(* Logix 5000 project; controller PLC_ABB vendor 1 type 14 code 77 rev 20.11; software revision 20.00 *)

TASK MainTask (continuous, watchdog 500 ms) : MainProgram

MODULES
   Controller : vendor 1 type 14 code 77 (CompactLogixL32EController 0, rev 20.11)
      LocalENB : 1769-L32E Ethernet Port (CompactLogixL32Ethernet 1, rev 20.11)
         PLC_DC : 1769-L32E Ethernet Port (Ethernet 192.168.2.131, rev 20.1)
            PLC_DC_Controller : vendor 1 type 14 code 77 (CompactLogixL32EController 0, rev 20.1, $a7c5510e$ RPI 20 ms, $928fdd19$ RPI 20 ms, $93e49bd8$ RPI 20 ms)
         ABBDrive : ETHERNET-MODULE (Ethernet 192.168.2.40, rev 1.1, Output RPI 20 ms)
      Local : CompactBus (CompactVirtualAdapter 3, rev 20.11)
         IO_Digital_Module : vendor 1 type 7 code 66 (Compact 2, rev 2.1, Output RPI 20 ms)
         hartModule : vendor 58 type 10 code 4 (Compact 1, rev 3.1, Output RPI 80 ms)
END_MODULES

TYPE ABB_Read :
STRUCT
   Logic_Status_Word : LSW;
   RPM_Feedback : INT;
   RPM_Referencia : INT;
   Output_Power : REAL;
   BusDC : REAL;
   Output_Current : REAL;
   Output_Voltage : REAL;
   PF : REAL;
   Latest_Fault : INT;
   Accel : BOOL;
   Descell : BOOL;
   PercentTemperature : INT;
END_STRUCT
END_TYPE

TYPE ABB_Write :
STRUCT
   RPM_Reference : INT;
   Run_Forward : BOOL;
   Run_Reverse : BOOL;
   Reset_Fault : BOOL;
END_STRUCT
END_TYPE

TYPE ComandVSD :
STRUCT
   start : BOOL;
   stop : BOOL;
   reset : BOOL;
   referencia : REAL;
   direction : BOOL;
END_STRUCT
END_TYPE

TYPE Dinagrama :
STRUCT
   vPotencia : REAL[500];
   vCarga : REAL[500];
   vPosicion : REAL[500];
   vProximetro : DINT[500];
   NumeroMuestras : INT;
   enabled : BOOL;
   captura : BOOL;
   resetVector : BOOL;
   vEmptyREAL : REAL[500];
   vEmptyINT : DINT[500];
   tMuestreo : REAL;
END_STRUCT
END_TYPE

TYPE ethImplicitRead :
STRUCT
   Enabled : BOOL;
   Done : BOOL;
   Error : BOOL;
   Value : DINT;
   instance : DINT;
   atribute : INT;
END_STRUCT
END_TYPE

TYPE ethImplicitWrite :
STRUCT
   Enabled : BOOL;
   Done : BOOL;
   ERR : BOOL;
   Value : DINT;
   Instance : DINT;
   Atribute : INT;
   clase : INT;
END_STRUCT
END_TYPE

TYPE LSW :
STRUCT
   Faulted : BOOL;
   Warning : BOOL;
   RunForward : BOOL;
   RunReverse : BOOL;
   Ready : BOOL;
   RemoteRef : BOOL;
   RemoteCrtl : BOOL;
   AtSpeed : BOOL;
END_STRUCT
END_TYPE

TYPE SWC :
STRUCT
   comand : ComandVSD;
   Dinagrama : Dinagrama;
   entradasDigitales : INT;
   salidasDigitales : INT;
   entradasAnalogas : REAL[4];
   salidasAnalogas : REAL[4];
   ABBRead : ABB_Read;
   etheWrite : ethImplicitWrite;
   etheRead : ethImplicitRead;
END_STRUCT
END_TYPE

TYPE VSD :
STRUCT
   LogicCommand_Start : BOOL;
   LogicCommand_Stop : BOOL;
   LogicCommand_ClearFaults : BOOL;
   LogicCommand_Forward : BOOL;
   LogicCommand_Reverse : BOOL;
   Reference : REAL;
END_STRUCT
END_TYPE

VAR_GLOBAL   (* controller tags *)
   ABB_GetAtt_Value : DINT := 7500;
   ABB_GetMsg : MESSAGE;
        MessageParameters(ServiceCode := 16#000e, DestinationTag := ABB_GetAtt_Value, ...)
   ABB_Input : ABB_Read := (Logic_Status_Word.Ready := 1, Logic_Status_Word.RemoteRef := 1, Logic_Status_Word.RemoteCrtl := 1, RPM_Referencia := 180, Output_Power := 5.8945793e-37, BusDC := 678.1, Latest_Fault := 8976, PercentTemperature := 20);
   ABB_Msg_SetValue : DINT := 60000;
   ABB_Output : ABB_Write := (RPM_Reference := 180);
   ABB_SetMsg : MESSAGE;
        MessageParameters(ServiceCode := 16#0010, LocalElement := ABB_Msg_SetValue, ...)
   Proximetro : BOOL;
   SRP_Displacement_Actual : REAL := 0.643343;
   SRP_Load_Actual : REAL := 9.741267;
   SRP_SimActualStroke : DINT := 1;
   SWC : SWC := (comand.referencia := 180.0, comand.direction := 1, Dinagrama.vPotencia[0] := 5.890374e-37, Dinagrama.vPotencia[1] := 5.890374e-37, Dinagrama.vPotencia[2] := 5.890374e-37, Dinagrama.vPotencia[3] := 5.890374e-37, Dinagrama.vPotencia[4] := 5.890374e-37, Dinagrama.vPotencia[5] := 5.890374e-37, Dinagrama.vPotencia[6] := 5.890374e-37, Dinagrama.vPotencia[7] := 5.890374e-37, Dinagrama.vPotencia[8] := 5.890374e-37, Dinagrama.vPotencia[9] := 5.890374e-37, Dinagrama.vPotencia[10] := 5.890374e-37, Dinagrama.vPotencia[11] := 5.890374e-37, Dinagrama.vPotencia[12] := 5.890374e-37, Dinagrama.vPotencia[13] := 5.890374e-37, Dinagrama.vPotencia[14] := 5.890374e-37, Dinagrama.vPotencia[15] := 5.890374e-37, Dinagrama.vPotencia[16] := 5.890374e-37, Dinagrama.vPotencia[17] := 5.890374e-37, Dinagrama.vPotencia[18] := 5.890374e-37, Dinagrama.vPotencia[19] := 5.890374e-37, Dinagrama.vPotencia[20] := 5.890374e-37, Dinagrama.vPotencia[21] := 5.890374e-37, Dinagrama.vPotencia[22] := 5.890374e-37, Dinagrama.vPotencia[23] := 5.890374e-37, Dinagrama.vPotencia[24] := 5.890374e-37, Dinagrama.vPotencia[25] := 5.890374e-37, Dinagrama.vPotencia[26] := 5.890374e-37, Dinagrama.vPotencia[27] := 5.890374e-37, Dinagrama.vPotencia[28] := 5.890374e-37, Dinagrama.vPotencia[29] := 5.890374e-37, Dinagrama.vPotencia[30] := 5.890374e-37, Dinagrama.vPotencia[31] := 5.890374e-37, Dinagrama.vPotencia[32] := 5.890374e-37, Dinagrama.vPotencia[33] := 5.890374e-37, Dinagrama.vPotencia[34] := 5.890374e-37, Dinagrama.vPotencia[35] := 5.890374e-37, Dinagrama.vPotencia[36] := 5.890374e-37, Dinagrama.vPotencia[37] := 5.890374e-37, Dinagrama.vPotencia[38] := 5.890374e-37, Dinagrama.vPotencia[39] := 5.890374e-37, Dinagrama.vPotencia[40] := 5.890374e-37, Dinagrama.vPotencia[41] := 5.890374e-37, Dinagrama.vPotencia[42] := 5.890374e-37, Dinagrama.vPotencia[43] := 5.890374e-37, Dinagrama.vPotencia[44] := 5.890374e-37, Dinagrama.vPotencia[45] := 5.890374e-37, Dinagrama.vPotencia[46] := 5.890374e-37, Dinagrama.vPotencia[47] := 5.890374e-37, Dinagrama.vPotencia[48] := 5.890374e-37, Dinagrama.vPotencia[49] := 5.890374e-37, Dinagrama.vPotencia[50] := 5.890374e-37, Dinagrama.vPotencia[51] := 5.890374e-37, Dinagrama.vPotencia[52] := 5.890374e-37, Dinagrama.vPotencia[53] := 5.890374e-37, Dinagrama.vPotencia[54] := 5.890374e-37, Dinagrama.vPotencia[55] := 5.890374e-37, Dinagrama.vPotencia[56] := 5.890374e-37, Dinagrama.vPotencia[57] := 5.890374e-37,
        Dinagrama.vPotencia[58] := 5.890374e-37, Dinagrama.vPotencia[59] := 5.890374e-37, Dinagrama.vPotencia[60] := 5.890374e-37, Dinagrama.vPotencia[61] := 5.890374e-37, Dinagrama.vPotencia[62] := 5.890374e-37, Dinagrama.vPotencia[63] := 5.890374e-37, Dinagrama.vPotencia[64] := 5.890374e-37, Dinagrama.vPotencia[65] := 5.890374e-37, Dinagrama.vPotencia[66] := 5.890374e-37, Dinagrama.vPotencia[67] := 5.890374e-37, Dinagrama.vPotencia[68] := 5.890374e-37, Dinagrama.vPotencia[69] := 5.890374e-37, Dinagrama.vPotencia[70] := 5.890374e-37, Dinagrama.vPotencia[71] := 5.890374e-37, Dinagrama.vPotencia[72] := 5.890374e-37, Dinagrama.vPotencia[73] := 5.890374e-37, Dinagrama.vPotencia[74] := 5.890374e-37, Dinagrama.vPotencia[75] := 5.890374e-37, Dinagrama.vPotencia[76] := 5.890374e-37, Dinagrama.vPotencia[77] := 5.890374e-37, Dinagrama.vPotencia[78] := 5.890374e-37, Dinagrama.vPotencia[79] := 5.890374e-37, Dinagrama.vPotencia[80] := 5.890374e-37, Dinagrama.vPotencia[81] := 5.890374e-37, Dinagrama.vPotencia[82] := 5.890374e-37, Dinagrama.vPotencia[83] := 5.890374e-37, Dinagrama.vPotencia[84] := 5.890374e-37, Dinagrama.vPotencia[85] := 5.890374e-37, Dinagrama.vPotencia[86] := 5.890374e-37, Dinagrama.vPotencia[87] := 5.890374e-37, Dinagrama.vPotencia[88] := 5.890374e-37, Dinagrama.vPotencia[89] := 5.890374e-37, Dinagrama.vPotencia[90] := 5.890374e-37, Dinagrama.vPotencia[91] := 5.890374e-37, Dinagrama.vPotencia[92] := 5.890374e-37, Dinagrama.vPotencia[93] := 5.890374e-37, Dinagrama.vPotencia[94] := 5.890374e-37, Dinagrama.vPotencia[95] := 5.890374e-37, Dinagrama.vPotencia[96] := 5.890374e-37, Dinagrama.vPotencia[97] := 5.890374e-37, Dinagrama.vPotencia[98] := 5.890374e-37, Dinagrama.vPotencia[99] := 5.890374e-37, Dinagrama.vPotencia[100] := 5.890374e-37, Dinagrama.vPotencia[101] := 5.890374e-37, Dinagrama.vPotencia[102] := 5.890374e-37, Dinagrama.vPotencia[103] := 5.890374e-37, Dinagrama.vPotencia[104] := 5.890374e-37, Dinagrama.vPotencia[105] := 5.890374e-37, Dinagrama.vPotencia[106] := 5.890374e-37, Dinagrama.vPotencia[107] := 5.890374e-37, Dinagrama.vPotencia[108] := 5.890374e-37, Dinagrama.vPotencia[109] := 5.890374e-37, Dinagrama.vPotencia[110] := 5.890374e-37, Dinagrama.vPotencia[111] := 5.890374e-37, Dinagrama.vPotencia[112] := 5.890374e-37, Dinagrama.vPotencia[113] := 5.890374e-37, Dinagrama.vPotencia[114] := 5.890374e-37, Dinagrama.vPotencia[115] := 5.890374e-37, Dinagrama.vPotencia[116] := 5.890374e-37, Dinagrama.vPotencia[117] := 5.890374e-37,
        Dinagrama.vPotencia[118] := 5.890374e-37, Dinagrama.vPotencia[119] := 5.890374e-37, Dinagrama.vPotencia[120] := 5.890374e-37, Dinagrama.vPotencia[121] := 5.890374e-37, Dinagrama.vPotencia[122] := 5.890374e-37, Dinagrama.vPotencia[123] := 5.890374e-37, Dinagrama.vPotencia[124] := 5.890374e-37, Dinagrama.vPotencia[125] := 5.890374e-37, Dinagrama.vPotencia[126] := 5.890374e-37, Dinagrama.vPotencia[127] := 5.890374e-37, Dinagrama.vPotencia[128] := 5.890374e-37, Dinagrama.vPotencia[129] := 5.890374e-37, Dinagrama.vPotencia[130] := 5.890374e-37, Dinagrama.vPotencia[131] := 5.890374e-37, Dinagrama.vPotencia[132] := 5.890374e-37, Dinagrama.vPotencia[133] := 5.890374e-37, Dinagrama.vPotencia[134] := 5.890374e-37, Dinagrama.vPotencia[135] := 5.890374e-37, Dinagrama.vPotencia[136] := 5.890374e-37, Dinagrama.vPotencia[137] := 5.890374e-37, Dinagrama.vPotencia[138] := 5.890374e-37, Dinagrama.vPotencia[139] := 5.890374e-37, Dinagrama.vPotencia[140] := 5.890374e-37, Dinagrama.vPotencia[141] := 5.890374e-37, Dinagrama.vPotencia[142] := 5.8988127e-37, Dinagrama.vCarga[0] := 9.6614, Dinagrama.vCarga[1] := 9.7812, Dinagrama.vCarga[2] := 9.711983, Dinagrama.vCarga[3] := 9.725293, Dinagrama.vCarga[4] := 9.842433, Dinagrama.vCarga[5] := 9.70932, Dinagrama.vCarga[6] := 9.69601, Dinagrama.vCarga[7] := 9.7306185, Dinagrama.vCarga[8] := 9.586858, Dinagrama.vCarga[9] := 9.751916, Dinagrama.vCarga[10] := 10.223133, Dinagrama.vCarga[11] := 10.473384, Dinagrama.vCarga[12] := 10.633119, Dinagrama.vCarga[13] := 10.856748, Dinagrama.vCarga[14] := 11.029794, Dinagrama.vCarga[15] := 11.220809, Dinagrama.vCarga[16] := 11.419147, Dinagrama.vCarga[17] := 11.515653, Dinagrama.vCarga[18] := 11.655421, Dinagrama.vCarga[19] := 11.805838, Dinagrama.vCarga[20] := 11.900348, Dinagrama.vCarga[21] := 11.940947, Dinagrama.vCarga[22] := 11.73795, Dinagrama.vCarga[23] := 11.4471, Dinagrama.vCarga[24] := 11.15625, Dinagrama.vCarga[25] := 10.976548, Dinagrama.vCarga[26] := 10.774218, Dinagrama.vCarga[27] := 10.571887, Dinagrama.vCarga[28] := 10.393517, Dinagrama.vCarga[29] := 10.257743, Dinagrama.vCarga[30] := 10.105995, Dinagrama.vCarga[31] := 10.018141, Dinagrama.vCarga[32] := 9.762565, Dinagrama.vCarga[33] := 9.634777, Dinagrama.vCarga[34] := 9.706658,
        Dinagrama.vCarga[35] := 9.826459, Dinagrama.vCarga[36] := 10.050088, Dinagrama.vCarga[37] := 10.177875, Dinagrama.vCarga[38] := 10.321636, Dinagrama.vCarga[39] := 10.409491, Dinagrama.vCarga[40] := 10.417477, Dinagrama.vCarga[41] := 10.401504, Dinagrama.vCarga[42] := 10.518642, Dinagrama.vCarga[43] := 10.481371, Dinagrama.vCarga[44] := 10.476047, Dinagrama.vCarga[45] := 10.63312, Dinagrama.vCarga[46] := 10.715649, Dinagrama.vCarga[47] := 10.476047, Dinagrama.vCarga[48] := 10.17255, Dinagrama.vCarga[49] := 9.970221, Dinagrama.vCarga[50] := 9.850419, Dinagrama.vCarga[51] := 9.608155, Dinagrama.vCarga[52] := 9.397838, Dinagrama.vCarga[53] := 9.405825, Dinagrama.vCarga[54] := 9.34193, Dinagrama.vCarga[55] := 9.131613, Dinagrama.vCarga[56] := 9.049084, Dinagrama.vCarga[57] := 9.08103, Dinagrama.vCarga[58] := 8.9266205, Dinagrama.vCarga[59] := 8.873376, Dinagrama.vCarga[60] := 9.155573, Dinagrama.vCarga[61] := 9.427122, Dinagrama.vCarga[62] := 9.549585, Dinagrama.vCarga[63] := 9.682697, Dinagrama.vCarga[64] := 9.906326, Dinagrama.vCarga[65] := 10.012816, Dinagrama.vCarga[66] := 9.980869, Dinagrama.vCarga[67] := 9.986194, Dinagrama.vCarga[68] := 9.962234, Dinagrama.vCarga[69] := 10.018141, Dinagrama.vCarga[70] := 10.042101, Dinagrama.vCarga[71] := 10.098008, Dinagrama.vCarga[72] := 10.193849, Dinagrama.vCarga[73] := 9.938273, Dinagrama.vCarga[74] := 9.618804, Dinagrama.vCarga[75] := 9.546924, Dinagrama.vCarga[76] := 9.55491, Dinagrama.vCarga[77] := 9.331282, Dinagrama.vCarga[78] := 9.171547, Dinagrama.vCarga[79] := 9.347255, Dinagrama.vCarga[80] := 9.219467, Dinagrama.vCarga[81] := 9.123626, Dinagrama.vCarga[82] := 9.18752, Dinagrama.vCarga[83] := 9.331282, Dinagrama.vCarga[84] := 9.166222, Dinagrama.vCarga[85] := 9.400499, Dinagrama.vCarga[86] := 9.565559, Dinagrama.vCarga[87] := 9.762566, Dinagrama.vCarga[88] := 9.688023, Dinagrama.vCarga[89] := 9.746592, Dinagrama.vCarga[90] := 9.885028, Dinagrama.vCarga[91] := 9.834445, Dinagrama.vCarga[92] := 9.634777, Dinagrama.vCarga[93] := 9.640101, Dinagrama.vCarga[94] := 9.624128,
        Dinagrama.vCarga[95] := 9.37654, Dinagrama.vCarga[96] := 9.184858, Dinagrama.vCarga[97] := 9.046422, Dinagrama.vCarga[98] := 8.665721, Dinagrama.vCarga[99] := 8.223788, Dinagrama.vCarga[100] := 7.936266, Dinagrama.vCarga[101] := 7.851074, Dinagrama.vCarga[102] := 7.6647167, Dinagrama.vCarga[103] := 7.398492, Dinagrama.vCarga[104] := 7.281353, Dinagrama.vCarga[105] := 7.238757, Dinagrama.vCarga[106] := 6.993831, Dinagrama.vCarga[107] := 6.706309, Dinagrama.vCarga[108] := 6.6796865, Dinagrama.vCarga[109] := 6.903315, Dinagrama.vCarga[110] := 7.1056457, Dinagrama.vCarga[111] := 7.3771944, Dinagrama.vCarga[112] := 7.773869, Dinagrama.vCarga[113] := 7.91763, Dinagrama.vCarga[114] := 7.909643, Dinagrama.vCarga[115] := 7.909643, Dinagrama.vCarga[116] := 8.300993, Dinagrama.vCarga[117] := 8.340926, Dinagrama.vCarga[118] := 8.460728, Dinagrama.vCarga[119] := 8.596502, Dinagrama.vCarga[120] := 8.804157, Dinagrama.vCarga[121] := 8.788184, Dinagrama.vCarga[122] := 8.77221, Dinagrama.vCarga[123] := 8.588515, Dinagrama.vCarga[124] := 8.420794, Dinagrama.vCarga[125] := 8.340927, Dinagrama.vCarga[126] := 8.468715, Dinagrama.vCarga[127] := 8.431443, Dinagrama.vCarga[128] := 8.476701, Dinagrama.vCarga[129] := 8.580528, Dinagrama.vCarga[130] := 8.497999, Dinagrama.vCarga[131] := 8.503324, Dinagrama.vCarga[132] := 8.575204, Dinagrama.vCarga[133] := 8.56988, Dinagrama.vCarga[134] := 8.631111, Dinagrama.vCarga[135] := 8.84409, Dinagrama.vCarga[136] := 9.081031, Dinagrama.vCarga[137] := 9.278037, Dinagrama.vCarga[138] := 9.325957, Dinagrama.vCarga[139] := 9.363229, Dinagrama.vCarga[140] := 9.618804, Dinagrama.vCarga[141] := 9.682698, Dinagrama.vCarga[142] := 9.682698, Dinagrama.vPosicion[0] := 0.0550175, Dinagrama.vPosicion[1] := 0.4084145, Dinagrama.vPosicion[2] := 0.8989175, Dinagrama.vPosicion[3] := 1.5143573, Dinagrama.vPosicion[4] := 2.2604218, Dinagrama.vPosicion[5] := 3.6340683, Dinagrama.vPosicion[6] := 4.147569, Dinagrama.vPosicion[7] := 5.2654533, Dinagrama.vPosicion[8] := 6.4805126, Dinagrama.vPosicion[9] := 7.78114, Dinagrama.vPosicion[10] := 9.158964, Dinagrama.vPosicion[11] := 10.613574,
        Dinagrama.vPosicion[12] := 12.155543, Dinagrama.vPosicion[13] := 13.778378, Dinagrama.vPosicion[14] := 15.740422, Dinagrama.vPosicion[15] := 17.481466, Dinagrama.vPosicion[16] := 19.2797, Dinagrama.vPosicion[17] := 21.118301, Dinagrama.vPosicion[18] := 22.99865, Dinagrama.vPosicion[19] := 24.928076, Dinagrama.vPosicion[20] := 26.89821, Dinagrama.vPosicion[21] := 28.908155, Dinagrama.vPosicion[22] := 30.958275, Dinagrama.vPosicion[23] := 33.057575, Dinagrama.vPosicion[24] := 35.193996, Dinagrama.vPosicion[25] := 37.35984, Dinagrama.vPosicion[26] := 39.561394, Dinagrama.vPosicion[27] := 41.798325, Dinagrama.vPosicion[28] := 44.44635, Dinagrama.vPosicion[29] := 46.757927, Dinagrama.vPosicion[30] := 49.113125, Dinagrama.vPosicion[31] := 50.300934, Dinagrama.vPosicion[32] := 53.71554, Dinagrama.vPosicion[33] := 56.007725, Dinagrama.vPosicion[34] := 58.29858, Dinagrama.vPosicion[35] := 59.435463, Dinagrama.vPosicion[36] := 61.651955, Dinagrama.vPosicion[37] := 64.96143, Dinagrama.vPosicion[38] := 67.1463, Dinagrama.vPosicion[39] := 69.277466, Dinagrama.vPosicion[40] := 70.327156, Dinagrama.vPosicion[41] := 72.39657, Dinagrama.vPosicion[42] := 74.763824, Dinagrama.vPosicion[43] := 77.68309, Dinagrama.vPosicion[44] := 78.62532, Dinagrama.vPosicion[45] := 80.46515, Dinagrama.vPosicion[46] := 82.25429, Dinagrama.vPosicion[47] := 83.99117, Dinagrama.vPosicion[48] := 85.65761, Dinagrama.vPosicion[49] := 87.23202, Dinagrama.vPosicion[50] := 88.73018, Dinagrama.vPosicion[51] := 90.154045, Dinagrama.vPosicion[52] := 91.48115, Dinagrama.vPosicion[53] := 92.103096, Dinagrama.vPosicion[54] := 93.858185, Dinagrama.vPosicion[55] := 94.9114, Dinagrama.vPosicion[56] := 96.00089, Dinagrama.vPosicion[57] := 96.84068, Dinagrama.vPosicion[58] := 97.581314, Dinagrama.vPosicion[59] := 98.21293, Dinagrama.vPosicion[60] := 98.7474, Dinagrama.vPosicion[61] := 99.18755, Dinagrama.vPosicion[62] := 99.53332, Dinagrama.vPosicion[63] := 99.672134, Dinagrama.vPosicion[64] := 99.935196, Dinagrama.vPosicion[65] := 99.99795, Dinagrama.vPosicion[66] := 99.96849, Dinagrama.vPosicion[67] := 99.8579, Dinagrama.vPosicion[68] := 99.76811, Dinagrama.vPosicion[69] := 99.35959, Dinagrama.vPosicion[70] := 98.93282, Dinagrama.vPosicion[71] := 98.72924,
        Dinagrama.vPosicion[72] := 98.26827, Dinagrama.vPosicion[73] := 97.74029, Dinagrama.vPosicion[74] := 97.14606, Dinagrama.vPosicion[75] := 96.147736, Dinagrama.vPosicion[76] := 95.795845, Dinagrama.vPosicion[77] := 95.004196, Dinagrama.vPosicion[78] := 94.16693, Dinagrama.vPosicion[79] := 93.305756, Dinagrama.vPosicion[80] := 91.870316, Dinagrama.vPosicion[81] := 91.377556, Dinagrama.vPosicion[82] := 90.37801, Dinagrama.vPosicion[83] := 89.32036, Dinagrama.vPosicion[84] := 87.43099, Dinagrama.vPosicion[85] := 86.2471, Dinagrama.vPosicion[86] := 85.63856, Dinagrama.vPosicion[87] := 84.37339, Dinagrama.vPosicion[88] := 83.06744, Dinagrama.vPosicion[89] := 81.722916, Dinagrama.vPosicion[90] := 79.59406, Dinagrama.vPosicion[91] := 78.86634, Dinagrama.vPosicion[92] := 77.38295, Dinagrama.vPosicion[93] := 75.84359, Dinagrama.vPosicion[94] := 74.24831, Dinagrama.vPosicion[95] := 72.63172, Dinagrama.vPosicion[96] := 70.97654, Dinagrama.vPosicion[97] := 69.25514, Dinagrama.vPosicion[98] := 67.223434, Dinagrama.vPosicion[99] := 65.45152, Dinagrama.vPosicion[100] := 63.614063, Dinagrama.vPosicion[101] := 61.744232, Dinagrama.vPosicion[102] := 59.862404, Dinagrama.vPosicion[103] := 57.93054, Dinagrama.vPosicion[104] := 55.949615, Dinagrama.vPosicion[105] := 53.960396, Dinagrama.vPosicion[106] := 51.950417, Dinagrama.vPosicion[107] := 49.88953, Dinagrama.vPosicion[108] := 47.795254, Dinagrama.vPosicion[109] := 45.690845, Dinagrama.vPosicion[110] := 43.56501, Dinagrama.vPosicion[111] := 41.413986, Dinagrama.vPosicion[112] := 38.891975, Dinagrama.vPosicion[113] := 36.722637, Dinagrama.vPosicion[114] := 34.528854, Dinagrama.vPosicion[115] := 33.423225, Dinagrama.vPosicion[116] := 30.155361, Dinagrama.vPosicion[117] := 27.987307, Dinagrama.vPosicion[118] := 25.821117, Dinagrama.vPosicion[119] := 24.743301, Dinagrama.vPosicion[120] := 22.634195, Dinagrama.vPosicion[121] := 20.581553, Dinagrama.vPosicion[122] := 17.632542, Dinagrama.vPosicion[123] := 15.761359, Dinagrama.vPosicion[124] := 14.84577, Dinagrama.vPosicion[125] := 13.085015, Dinagrama.vPosicion[126] := 11.154951, Dinagrama.vPosicion[127] := 8.857708, Dinagrama.vPosicion[128] := 8.136012, Dinagrama.vPosicion[129] := 6.7788615, Dinagrama.vPosicion[130] := 5.529149, Dinagrama.vPosicion[131] := 4.3940463,
        Dinagrama.vPosicion[132] := 2.945591, Dinagrama.vPosicion[133] := 2.520764, Dinagrama.vPosicion[134] := 1.7710685, Dinagrama.vPosicion[135] := 1.148738, Dinagrama.vPosicion[136] := 0.66532767, Dinagrama.vPosicion[137] := 0.31461334, Dinagrama.vPosicion[138] := 0.096083336, Dinagrama.vPosicion[139] := 0.009929333, Dinagrama.vPosicion[140] := 0.049646668, Dinagrama.vPosicion[141] := 0.059576, Dinagrama.vPosicion[142] := 0.059576, Dinagrama.vProximetro[0] := 1, Dinagrama.vProximetro[1] := 1, Dinagrama.vProximetro[2] := 1, Dinagrama.NumeroMuestras := 141, Dinagrama.tMuestreo := 0.05, entradasAnalogas[0] := 16.901644, entradasAnalogas[1] := 13.587194, entradasAnalogas[2] := 3.2056525, entradasAnalogas[3] := 3.2056525, ABBRead.Logic_Status_Word.Ready := 1, ABBRead.Logic_Status_Word.RemoteRef := 1, ABBRead.Logic_Status_Word.RemoteCrtl := 1, ABBRead.RPM_Referencia := 180, ABBRead.Output_Power := 5.8945793e-37, ABBRead.BusDC := 678.1, ABBRead.Latest_Fault := 8976, ABBRead.PercentTemperature := 20, etheWrite.Enabled := 1, etheWrite.ERR := 1, etheWrite.Value := 60000, etheWrite.Instance := 23, etheWrite.Atribute := 13, etheRead.Value := 7500, etheRead.instance := 99, etheRead.atribute := 10);
   Timmers : TIMER[10] := ([0].PRE := 43, [1].PRE := 828000, [1].ACC := 352537, [1].EN := 1, [1].TT := 1, [2].PRE := 500, [3].PRE := 1000, [4].PRE := 10000);
END_VAR

PROGRAM MainProgram   (* main routine R000_MainRoutine *)
VAR
   Captura : BOOL;
   contadorAux : ALIAS FOR counter[0].ACC;
   counter : COUNTER[10];
   Flag : BOOL;
   flagDesAcell : BOOL;
   myoneshot : BOOL[32] := ([0] := 1);
   Proximetro_Virtual : ALIAS FOR SRP_SimActualStroke;
   rpmFeedback : INT;
   SPM_Reference : REAL := 8.5;
   timer : TIMER[10] := ([0].PRE := 50);
END_VAR

ROUTINE R000_MainRoutine   (* ladder *)
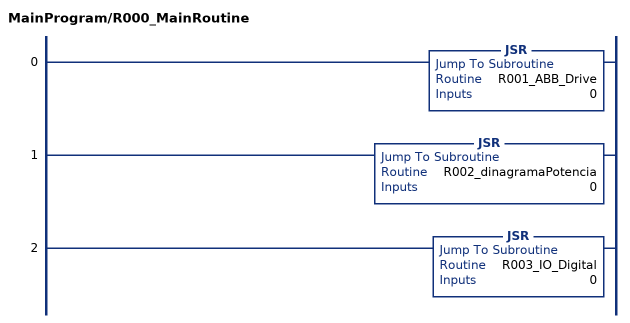
   0: JSR(R001_ABB_Drive,0);
   1: JSR(R002_dinagramaPotencia,0);
   2: JSR(R003_IO_Digital,0);
END_ROUTINE

ROUTINE R001_ABB_Drive   (* ladder *)
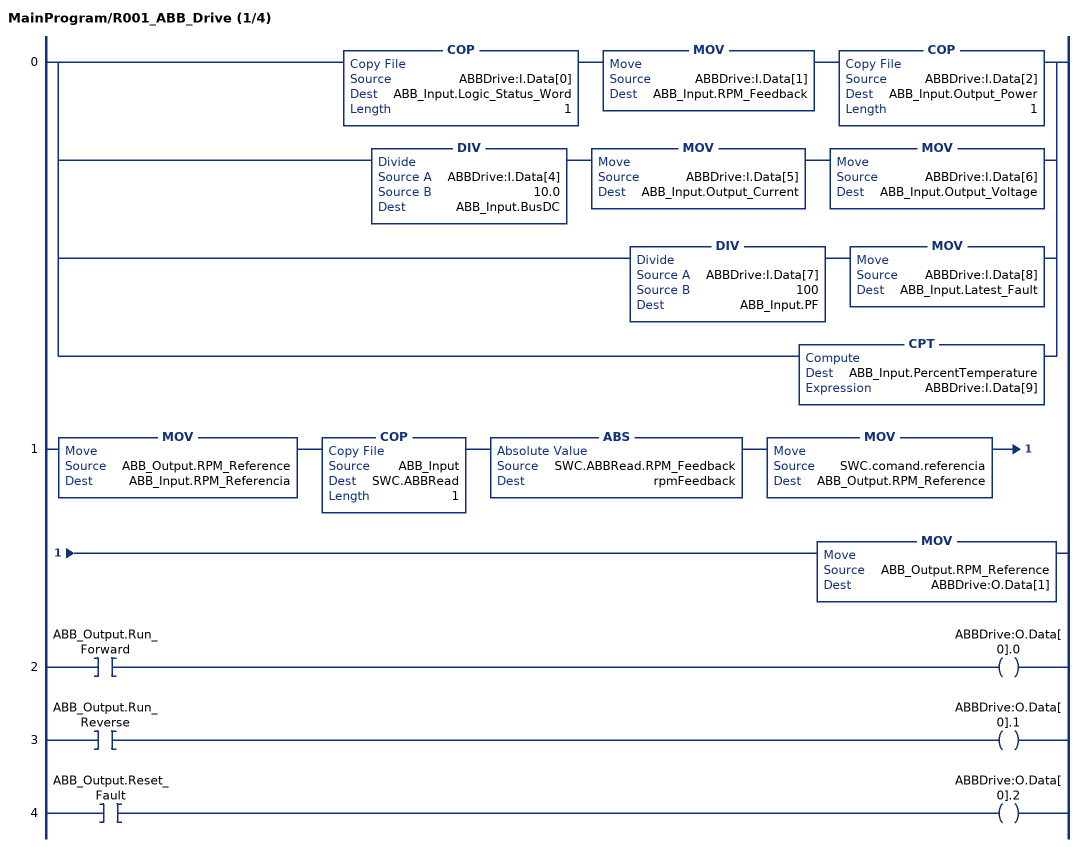
   0: [COP(ABBDrive:I.Data[0],ABB_Input.Logic_Status_Word,1) MOV(ABBDrive:I.Data[1],ABB_Input.RPM_Feedback) COP(ABBDrive:I.Data[2],ABB_Input.Output_Power,1) ,DIV(ABBDrive:I.Data[4],10.0,ABB_Input.BusDC) MOV(ABBDrive:I.Data[5],ABB_Input.Output_Current) MOV(ABBDrive:I.Data[6],ABB_Input.Output_Voltage) ,[DIV(ABBDrive:I.Data[7],100,ABB_Input.PF) MOV(ABBDrive:I.Data[8],ABB_Input.Latest_Fault) ,CPT(ABB_Input.PercentTemperature,ABBDrive:I.Data[9]) ] ];
   1: MOV(ABB_Output.RPM_Reference,ABB_Input.RPM_Referencia)COP(ABB_Input,SWC.ABBRead,1)ABS(SWC.ABBRead.RPM_Feedback,rpmFeedback)MOV(SWC.comand.referencia,ABB_Output.RPM_Reference)MOV(ABB_Output.RPM_Reference,ABBDrive:O.Data[1]);
   2: XIC(ABB_Output.Run_Forward)OTE(ABBDrive:O.Data[0].0);
   3: XIC(ABB_Output.Run_Reverse)OTE(ABBDrive:O.Data[0].1);
   4: XIC(ABB_Output.Reset_Fault)OTE(ABBDrive:O.Data[0].2);
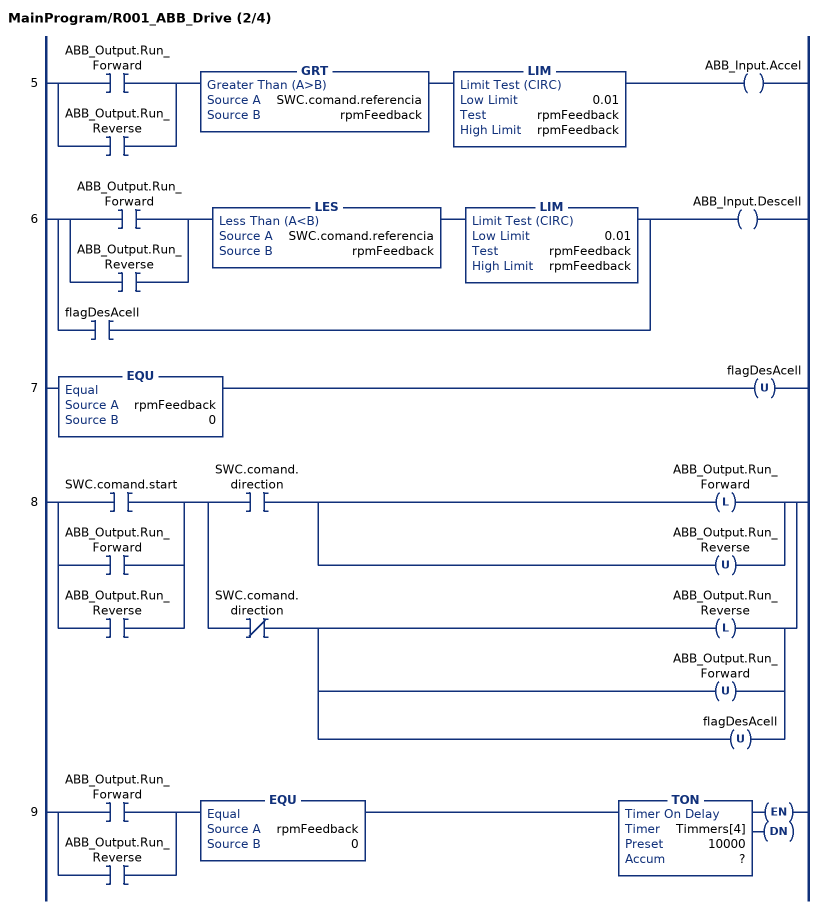
   5: [XIC(ABB_Output.Run_Forward) ,XIC(ABB_Output.Run_Reverse) ]GRT(SWC.comand.referencia,rpmFeedback)LIM(0.01,rpmFeedback,rpmFeedback)OTE(ABB_Input.Accel);
   6: [[XIC(ABB_Output.Run_Forward) ,XIC(ABB_Output.Run_Reverse) ] LES(SWC.comand.referencia,rpmFeedback) LIM(0.01,rpmFeedback,rpmFeedback) ,XIC(flagDesAcell) ]OTE(ABB_Input.Descell);
   7: EQU(rpmFeedback,0)OTU(flagDesAcell);
   8: [[XIC(SWC.comand.start) ,XIC(ABB_Output.Run_Forward) ] ,XIC(ABB_Output.Run_Reverse) ][XIC(SWC.comand.direction) [OTL(ABB_Output.Run_Forward) ,OTU(ABB_Output.Run_Reverse) ] ,XIO(SWC.comand.direction) [OTL(ABB_Output.Run_Reverse) ,[OTU(ABB_Output.Run_Forward) ,OTU(flagDesAcell) ] ] ];
   9: [XIC(ABB_Output.Run_Forward) ,XIC(ABB_Output.Run_Reverse) ]EQU(rpmFeedback,0)TON(Timmers[4],?,?);
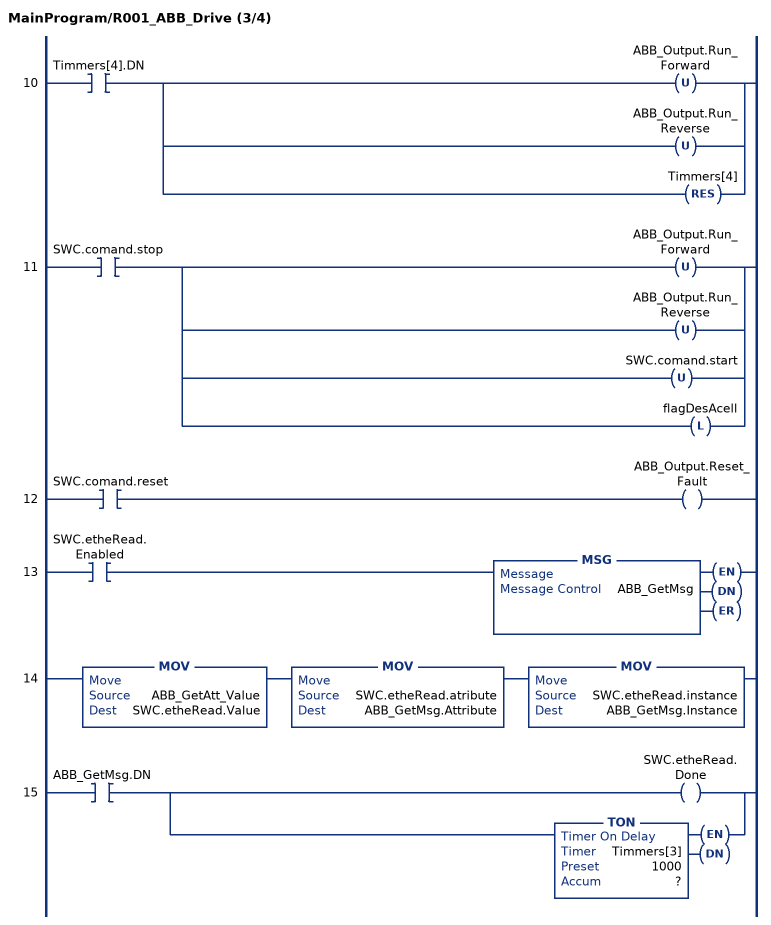
   10: XIC(Timmers[4].DN)[OTU(ABB_Output.Run_Forward) ,[OTU(ABB_Output.Run_Reverse) ,RES(Timmers[4]) ] ];
   11: XIC(SWC.comand.stop)[OTU(ABB_Output.Run_Forward) ,[OTU(ABB_Output.Run_Reverse) ,[OTU(SWC.comand.start) ,OTL(flagDesAcell) ] ] ];
   12: XIC(SWC.comand.reset)OTE(ABB_Output.Reset_Fault);
   13: XIC(SWC.etheRead.Enabled)MSG(ABB_GetMsg);
   14: MOV(ABB_GetAtt_Value,SWC.etheRead.Value)MOV(SWC.etheRead.atribute,ABB_GetMsg.Attribute)MOV(SWC.etheRead.instance,ABB_GetMsg.Instance);
   15: XIC(ABB_GetMsg.DN)[OTE(SWC.etheRead.Done) ,TON(Timmers[3],?,?) ];
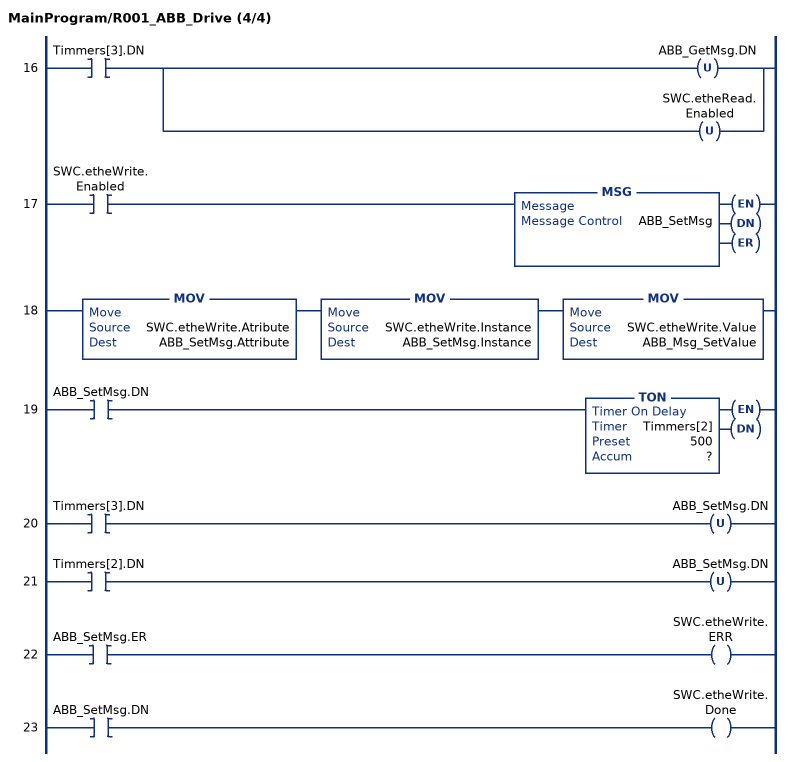
   16: XIC(Timmers[3].DN)[OTU(ABB_GetMsg.DN) ,OTU(SWC.etheRead.Enabled) ];
   17: XIC(SWC.etheWrite.Enabled)MSG(ABB_SetMsg);
   18: MOV(SWC.etheWrite.Atribute,ABB_SetMsg.Attribute)MOV(SWC.etheWrite.Instance,ABB_SetMsg.Instance)MOV(SWC.etheWrite.Value,ABB_Msg_SetValue);
   19: XIC(ABB_SetMsg.DN)TON(Timmers[2],?,?);
   20: XIC(Timmers[3].DN)OTU(ABB_SetMsg.DN);
   21: XIC(Timmers[2].DN)OTU(ABB_SetMsg.DN);
   22: XIC(ABB_SetMsg.ER)OTE(SWC.etheWrite.ERR);
   23: XIC(ABB_SetMsg.DN)OTE(SWC.etheWrite.Done);
END_ROUTINE

ROUTINE R002_dinagramaPotencia   (* ladder *)
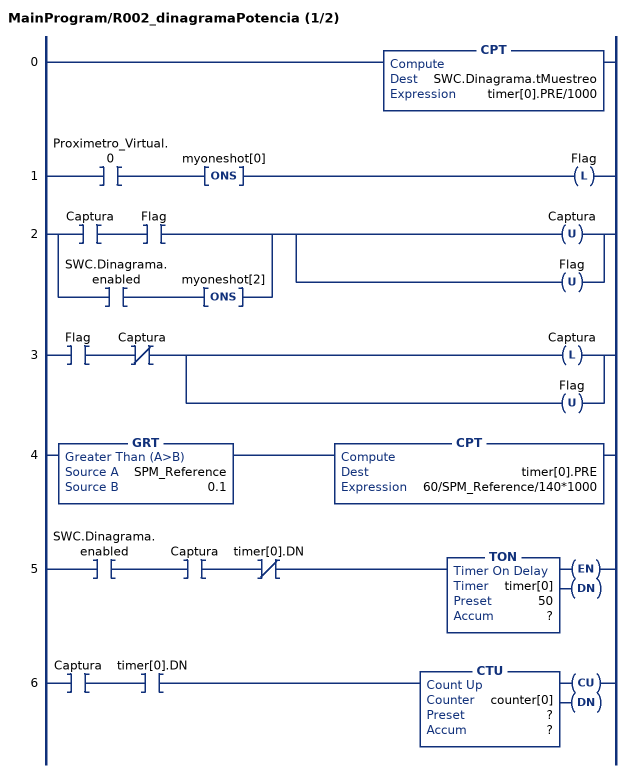
   0: CPT(SWC.Dinagrama.tMuestreo,timer[0].PRE/1000);
   1: XIC(Proximetro_Virtual.0)ONS(myoneshot[0])OTL(Flag);
   2: [XIC(Captura) XIC(Flag) ,XIC(SWC.Dinagrama.enabled) ONS(myoneshot[2]) ][OTU(Captura) ,OTU(Flag) ];
   3: XIC(Flag)XIO(Captura)[OTL(Captura) ,OTU(Flag) ];
   4: GRT(SPM_Reference,0.1)CPT(timer[0].PRE,60/SPM_Reference/140*1000);
   5: XIC(SWC.Dinagrama.enabled)XIC(Captura)XIO(timer[0].DN)TON(timer[0],?,?);
   6: XIC(Captura)XIC(timer[0].DN)CTU(counter[0],?,?);
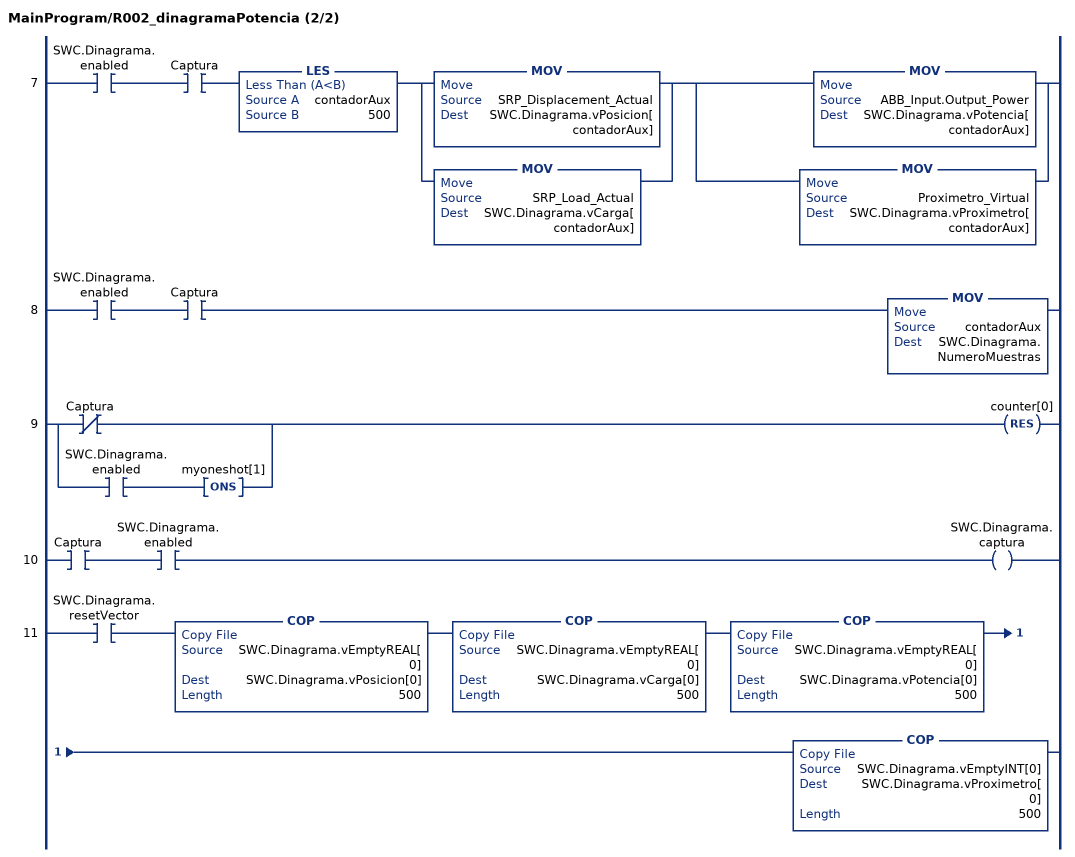
   7: XIC(SWC.Dinagrama.enabled)XIC(Captura)LES(contadorAux,500)[MOV(SRP_Displacement_Actual,SWC.Dinagrama.vPosicion[contadorAux]) ,MOV(SRP_Load_Actual,SWC.Dinagrama.vCarga[contadorAux]) ][MOV(ABB_Input.Output_Power,SWC.Dinagrama.vPotencia[contadorAux]) ,MOV(Proximetro_Virtual,SWC.Dinagrama.vProximetro[contadorAux]) ];
   8: XIC(SWC.Dinagrama.enabled)XIC(Captura)MOV(contadorAux,SWC.Dinagrama.NumeroMuestras);
   9: [XIO(Captura) ,XIC(SWC.Dinagrama.enabled) ONS(myoneshot[1]) ]RES(counter[0]);
   10: XIC(Captura)XIC(SWC.Dinagrama.enabled)OTE(SWC.Dinagrama.captura);
   11: XIC(SWC.Dinagrama.resetVector)COP(SWC.Dinagrama.vEmptyREAL[0],SWC.Dinagrama.vPosicion[0],500)COP(SWC.Dinagrama.vEmptyREAL[0],SWC.Dinagrama.vCarga[0],500)COP(SWC.Dinagrama.vEmptyREAL[0],SWC.Dinagrama.vPotencia[0],500)COP(SWC.Dinagrama.vEmptyINT[0],SWC.Dinagrama.vProximetro[0],500);
END_ROUTINE

ROUTINE R003_IO_Digital   (* ladder *)
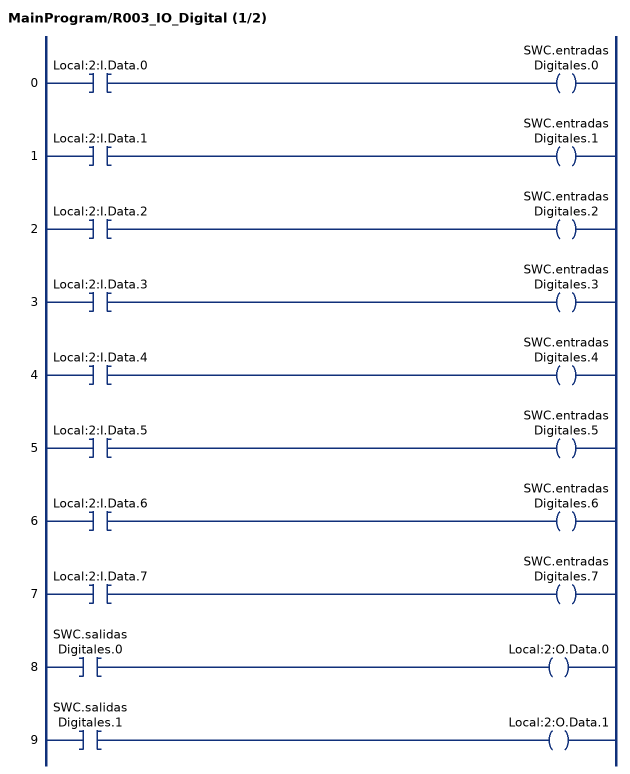
   0: XIC(Local:2:I.Data.0)OTE(SWC.entradasDigitales.0);
   1: XIC(Local:2:I.Data.1)OTE(SWC.entradasDigitales.1);
   2: XIC(Local:2:I.Data.2)OTE(SWC.entradasDigitales.2);
   3: XIC(Local:2:I.Data.3)OTE(SWC.entradasDigitales.3);
   4: XIC(Local:2:I.Data.4)OTE(SWC.entradasDigitales.4);
   5: XIC(Local:2:I.Data.5)OTE(SWC.entradasDigitales.5);
   6: XIC(Local:2:I.Data.6)OTE(SWC.entradasDigitales.6);
   7: XIC(Local:2:I.Data.7)OTE(SWC.entradasDigitales.7);
   8: XIC(SWC.salidasDigitales.0)OTE(Local:2:O.Data.0);
   9: XIC(SWC.salidasDigitales.1)OTE(Local:2:O.Data.1);
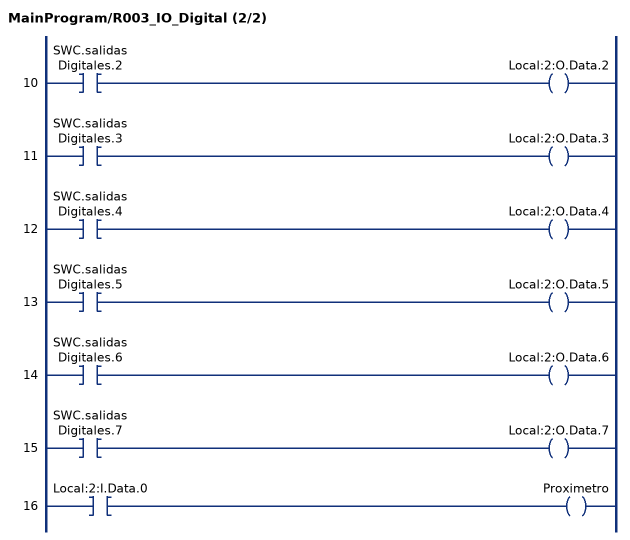
   10: XIC(SWC.salidasDigitales.2)OTE(Local:2:O.Data.2);
   11: XIC(SWC.salidasDigitales.3)OTE(Local:2:O.Data.3);
   12: XIC(SWC.salidasDigitales.4)OTE(Local:2:O.Data.4);
   13: XIC(SWC.salidasDigitales.5)OTE(Local:2:O.Data.5);
   14: XIC(SWC.salidasDigitales.6)OTE(Local:2:O.Data.6);
   15: XIC(SWC.salidasDigitales.7)OTE(Local:2:O.Data.7);
   16: XIC(Local:2:I.Data.0)OTE(Proximetro);
END_ROUTINE
END_PROGRAM
